ADAPTER aTest (* Adapter Interface *)
  (* Standard: 61499-1 *)
  (* Version 0.0, 10/1/2026, Schneider Electric *)
  PACKAGE Main;
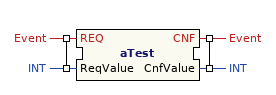
  EVENT_INPUT
    REQ WITH ReqValue; (* Request from Socket *)
  END_EVENT
  EVENT_OUTPUT
    CNF WITH CnfValue; (* Confirmation from Plug *)
  END_EVENT
  VAR_INPUT
    ReqValue : INT;
  END_VAR
  VAR_OUTPUT
    CnfValue : INT;
  END_VAR
  SERVICE SOCKET/PLUG
    SEQUENCE request_confirm
      SOCKET.REQ(REQD) -> PLUG.REQ(REQD);
      PLUG.CNF(CNFD) -> SOCKET.CNF(CNFD);
    END_SEQUENCE
    SEQUENCE indication_response
      PLUG.IND(INDD) -> SOCKET.IND(INDD);
      SOCKET.RSP(RSPD) -> PLUG.RSP(RSPD);
    END_SEQUENCE
  END_SERVICE
END_ADAPTER
